{attribute addProperty BoxType "EL2014-0000-0016"}
{attribute addProperty Id "Common_FaultAT %I*BOOL8117Overtemperature_DeviceAT %I*BOOL8118UndervoltageAT %I*BOOL8119Missing_VoltageAT %I*BOOL8120"}
{attribute addProperty CRC "120954638"}
{attribute addProperty SizeInBites "32"}
{attribute addProperty SizeInBytes "4"}
TYPE DIG_Inputs_Device_07359F0E :
STRUCT
	{attribute addProperty Name "Common_Fault"}
	Common_Fault AT %I* : BOOL;
	{attribute addProperty Name "Overtemperature_Device"}
	Overtemperature_Device AT %I* : BOOL;
	{attribute addProperty Name "Undervoltage"}
	Undervoltage AT %I* : BOOL;
	{attribute addProperty Name "Missing_Voltage"}
	Missing_Voltage AT %I* : BOOL;
END_STRUCT
END_TYPE

(* stored: Version 1.2.0.0, ProductVersion 3.1.4024.9
   DUT DIG_Inputs_Device_07359F0E: Id {e14c43cb-3c45-47d9-965e-23dc6aaaf3da} *)
